{attribute 'GeneratedUsingTerminal: ELM9410-0000-0016'}
{attribute addProperty BoxType "ELM9410-0000-0016"}
{attribute addProperty Id "ControlAT %Q*Control_EBEDCF761"}
{attribute addProperty CRC "3873896913"}
{attribute addProperty Size "1"}
TYPE MMS_Device_Outputs_E6E6F9D1 EXTENDS OutputBase_10CEE7DE :
STRUCT
	{attribute addProperty Name "Control"}
	Control AT %Q* : Control_EBEDCF76;
END_STRUCT
END_TYPE

(* stored: Version 1.2.0.0, ProductVersion 3.1.4024.9
   DUT MMS_Device_Outputs_E6E6F9D1: Id {ca7c9bc4-c06a-4cde-a066-f376722d9963} *)
